{attribute addProperty BoxType "ER6001-0002-0016"}
{attribute addProperty Id "COM_InputsAT %I*COM_Inputs_18212A5E192240COM_OutputsAT %Q*COM_Outputs_F536B385192240WcStateAT %I*WcState_98A4DF7520.250InfoDataAT %I*InfoData_BC63D37F80100"}
{attribute addProperty CRC "3759694539"}
{attribute addProperty SizeInBites "466"}
{attribute addProperty SizeInBytes "58.25"}
TYPE ER6001_79044676 :
STRUCT
	{attribute addProperty Name "COM_Inputs"}
	COM_Inputs : COM_Inputs_18212A5E;
	{attribute addProperty Name "COM_Outputs"}
	COM_Outputs : COM_Outputs_F536B385;
	{attribute addProperty Name "WcState"}
	WcState : WcState_98A4DF75;
	{attribute addProperty Name "InfoData"}
	InfoData : InfoData_BC63D37F;
END_STRUCT
END_TYPE

(* stored: Version 1.2.0.0, ProductVersion 3.1.4024.9
   DUT ER6001_79044676: Id {c5ce9c29-bd2c-4b69-b6f9-6567aba5bfba} *)
